Yaskawa INFORM job: OPDR3B.JBI

/JOB
//NAME OPDR3B
//POS
///NPOS 0,0,0,0,0,0
//INST
///DATE 2023/05/15 22:23
///ATTR SC,RW
///GROUP1 RB1
NOP
SET I001 1
' I001 = 1
SET I002 2
' I002 = 2
SET I003 3
' I003 = 3
SET I004 4
' I004 = 4
SET I005 5
' I005 = 5
SET I006 6
' I006 = 6
SET I007 7
' I007 = 7
SET I008 8
' I008 = 8
SET I009 9
' I009 = 9
SET I010 10
' I010 = 10
SET I011 11
' I011 = 11
SET I012 12
' I012 = 12
SET I021 I001
' I021 = I001 = 1
MUL I021 I002
' I021 = I021 * I002 = 1 * 2 = 2
SET I023 I003
' I023 = I003 = 3
MUL I023 I004
' I023 = I023 * I004 = 3 * 4 = 12
SET I031 I021
' I031 = I021 = 2
SET I032 I023
' I032 = I023 = 12
SUB I031 I032
' I031 = I031 - I032 = 2 - 12 = -10
ADD I031 I005
' I031 = I031 + I005 = -10 + 5 = -5
DIV I031 I006
' I031 = I031 / I006 = -5 / 6 = 0 (integer division)
SET I000 I031
' I000 = I031 = 0
SET D011 11
' D011 = 11.0
SET D012 12
' D012 = 12.0
SET D013 13
' D013 = 13.0
SET D014 14
' D014 = 14.0
SET D111 D011
' D111 = D011 = 11.0
SET D112 D012
' D112 = D012 = 12.0
DIV D111 D112
' D111 = D111 / D112 = 11.0 / 12.0
' = 0.9166666666666666 (floating-point division)
MUL D111 D014
' D111 = D111 * D014
' = 0.9166666666666666 * 14.0 = 12.833333333333332
SET D113 D013
' D113 = D013 = 13.0
DIV D113 D112
' D113 = D113 / D112 = 13.0 / 12.0
' = 1.0833333333333333 (floating-point division)
SUB D111 D113
' D111 = D111 - D113
' = 12.833333333333332 - 1.0833333333333333 = 11.75
SET D161 8
' D161 = 8.0
MUL D111 D161
' D111 = D111 * D161 = 11.75 * 8.0 = 94.0
SET I010 D111
' I010 = D111 = 94.0 (converted to an integer)
END
